FUNCTION ARR08X_TO_ST08X (* this Function takes a a 8-BOOL Array and makes a 8-BOOL Struct *)
  (* Standard: 61499-1; Description: Copyright (c) 2024 HR Agrartechnik GmbH This program and the accompanying materials are made available under the terms of the Eclipse Public License 2.0 which is available at https://www.eclipse.org/legal/epl-2.0/ SPDX-License-Identifier: EPL-2.0 *)
  (* Version 1.0, 2024-02-22, Franz Höpfinger, HR Agrartechnik GmbH *)
  PACKAGE logiBUS::utils::conversion::str::converting;
  IMPORT logiBUS::utils::conversion::types::ST08X;
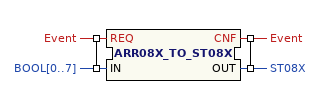
  EVENT_INPUT
    REQ WITH IN;
  END_EVENT
  EVENT_OUTPUT
    CNF WITH OUT;
  END_EVENT
  VAR_INPUT
    IN : ARRAY [0..7] OF BOOL; (* ARR08X Input *)
  END_VAR
  VAR_OUTPUT
    OUT : logiBUS::utils::conversion::types::ST08X; (* ST08X Output *)
  END_VAR
  BODY IN ST:
PACKAGE logiBUS::utils::conversion::str::converting;

IMPORT logiBUS::utils::conversion::types::ST08X;

(* this Function takes a a 8-BOOL Array and makes a 8-BOOL Struct *)
FUNCTION ARR08X_TO_ST08X

VAR_INPUT
	IN : ARRAY[0..7] OF BOOL; // ARR08X Input
END_VAR

VAR_OUTPUT
	OUT : ST08X; // ST08X Output
END_VAR

OUT.X_00 := IN[0];
OUT.X_01 := IN[1];
OUT.X_02 := IN[2];
OUT.X_03 := IN[3];
OUT.X_04 := IN[4];
OUT.X_05 := IN[5];
OUT.X_06 := IN[6];
OUT.X_07 := IN[7];

END_FUNCTION
  END_BODY
END_FUNCTION
